VAR_GLOBAL
	{attribute 'pytmc' :=' pv: EM1K0:GMD:OVERRIDE_VAC '}
	xSystemOverrideMode : BOOL; (* Global system override for the prototype section*)
	
	{attribute 'pytmc' :=' pv: EM1K0:GMD:AUTO_VVC_40 '}
	bAutoVVC40 : BOOL := False;
	
	{attribute 'pytmc' := '
	pv: EM1K0:GMD:GAS_TYPE ;
	type: mbbi ;
	field: ZRST none ;
	field: ONST Neon;
	field: TWST Argon ;
	field: THST Krypton ;
	field: FRST Xenon ;
	io: i
	'}
	SelectedGas: E_GasType;
	
		// Purge COMMANDS FROM epics
	//pragma
	{attribute 'pytmc' :=' pv: EM1K0:GMD:Purge_SW'}
	bStartPurge_sw : BOOL :=false;
	{attribute 'pytmc' :=' pv: EM1K0:GMD:Purge_Active'}
	bPurgeActive : BOOL:=false;
	{attribute 'pytmc' :=' pv: EM1K0:GMD:PurgeDone'}
	bPurgeDone : BOOL :=false;
	
	fbLogHandler : FB_LogHandler;
END_VAR

(* stored: Version 1.1.0.1, ProductVersion 3.1.4022.18
   GVL GVL_VARIABLES: Id {f5eb425e-877f-4a98-b4fc-8b7970a753e9} *)
